// TIA Portal V19 export
DATA_BLOCK "SimulationData"   // DB58
// stored: MemoryReserve 100, Namespace Unit3
BEGIN
END_DATA_BLOCK
